FUNCTION_BLOCK FB_HomeReadNcVelocities
VAR_INPUT
    bReset: BOOL;
    bExecute: BOOL;
END_VAR
VAR_IN_OUT
    Axis: AXIS_REF;
END_VAR
VAR_OUTPUT
    bBusy: BOOL;
    bDone: BOOL;
    bError: BOOL;
    nErrorId: UDINT;
    fVelocityToCam: LREAL;
    fVelocityFromCam: LREAL;
END_VAR
VAR
    fbReadVelocityToCam: FB_ReadFloatParameter;
    fbReadVelocityFromCam: FB_ReadFloatParameter;
END_VAR

fbReadVelocityToCam(Axis:= Axis);
fbReadVelocityFromCam(Axis:= Axis);

IF bReset THEN
    bError := FALSE;
    nErrorId := 0;
END_IF

fbReadVelocityToCam.bExecute := bExecute;
fbReadVelocityToCam.nDeviceGroup := 16#4000;
fbReadVelocityToCam.nIndexOffset := 16#6;

fbReadVelocityFromCam.bExecute := bExecute;
fbReadVelocityFromCam.nDeviceGroup := 16#4000;
fbReadVelocityFromCam.nIndexOffset := 16#7;

fVelocityToCam := fbReadVelocityToCam.nData;
fVelocityFromCam := fbReadVelocityFromCam.nData;

bBusy := fbReadVelocityFromCam.bBusy OR fbReadVelocityToCam.bBusy;
bDone := fbReadVelocityFromCam.bDone AND fbReadVelocityToCam.bDone AND bExecute;
bError := fbReadVelocityToCam.bError OR fbReadVelocityFromCam.bError;

IF fbReadVelocityToCam.bError THEN
  nErrorId := fbReadVelocityToCam.nErrorId;
ELSIF fbReadVelocityFromCam.bError THEN
  nErrorId := fbReadVelocityFromCam.nErrorId;
END_IF

END_FUNCTION_BLOCK

(* stored: Version 1.1.0.1, ProductVersion 3.1.4024.0
   POU FB_HomeReadNcVelocities: Id {a78232f2-2338-46fa-908d-fbea8ac2e783}, SpecialFunc None *)
